{attribute 'GeneratedUsingTerminal: EK1100-0000-0018'}
{attribute addProperty BoxType "EK1100-0000-0018"}
{attribute addProperty Id "Beckhoff_EPP7xxxEK1122Beckhoff_EPP7xxxEK1122_4AE68EFB550"}
{attribute addProperty CRC "650532054"}
{attribute addProperty Size "550"}
TYPE Beckhoff_EPP7xxx_26C654D6 EXTENDS EK1100_1FC0878B :
STRUCT
	{attribute addProperty Name "Beckhoff_EPP7xxxEK1122"}
	Beckhoff_EPP7xxxEK1122 : Beckhoff_EPP7xxxEK1122_4AE68EFB;
END_STRUCT
END_TYPE

(* stored: Version 1.2.0.0, ProductVersion 3.1.4024.9
   DUT Beckhoff_EPP7xxx_26C654D6: Id {ae16a1a4-791b-42aa-8180-21414a20b7e1} *)
